// TIA Portal V16 export
// export: Created 2021-09-08T12:46:08.2210829Z, ExportSetting WithDefaults, DisplayName Totally Integrated Automation Portal, DisplayVersion V16 Update 3, DisplayName TIA Portal Version Control Interface, DisplayVersion V16 Update 2, DisplayName TIA Portal Openness, DisplayVersion V16 Update 3, DisplayName TIA Portal Teamcenter Gateway, DisplayVersion V16, DisplayName STEP 7 Professional, DisplayVersion V16 Update 3, DisplayName STEP 7 Safety, DisplayVersion V16, DisplayName WinCC Advanced, DisplayVersion V16 Update 3
FUNCTION_BLOCK "noPulseTOF"   // FB15, FBD
{ S7_Optimized_Access := 'TRUE' }
VERSION : 0.1
// stored: AutoNumber true, IsIECCheckEnabled false, IsRetainMemResEnabled false, MemoryReserve 100, SetENOAutomatically false, UDAEnableTagReadback false
   VAR_INPUT
      pulse : Bool;
      timeSP_sec : Real;
      reset : Bool;
   END_VAR
   VAR_OUTPUT
      out : Bool;
   END_VAR
   VAR
      curTime : Real;
      nTrig : Bool;
      pTirg : Bool;
   END_VAR
   VAR_TEMP   // added for the SCL form of the ladder/FBD networks
      _w1 : Bool;
      _w2 : Bool;
   END_VAR
BEGIN

REGION Network 1: Увеличение времени
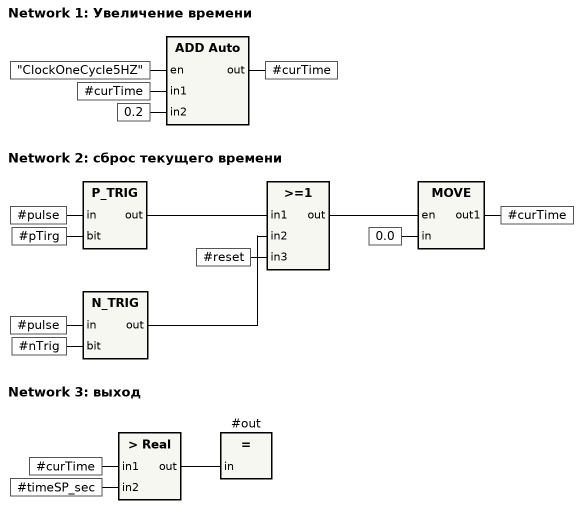
   IF "ClockOneCycle5HZ" THEN #curTime := #curTime + 0.2; END_IF;
END_REGION

REGION Network 2: сброс текущего времени
   #_w1 := #pulse AND NOT #pTirg;   // rising edge
   #pTirg := #pulse;
   #_w2 := NOT #pulse AND #nTrig;   // falling edge
   #nTrig := #pulse;
   IF #_w1 OR #_w2 OR #reset THEN #curTime := 0.0; END_IF;
END_REGION

REGION Network 3: выход
   #out := #curTime > #timeSP_sec;
END_REGION
END_FUNCTION_BLOCK
